METHOD SetUserFrame : BOOL
VAR_INPUT
	Frame	: ST_CartesianPoint;
END_VAR
VAR_OUTPUT
	task	: RoboConnect.I_Task;
END_VAR
VAR 
  commandString : T_Maxstring; 
  
  tableString : STRING := '{,,,,,}';
END_VAR
// TODO better ways of doing this.
tableString := INSERT(tableString, LREAL_TO_STRING(Frame.c),6);
tableString := INSERT(tableString, LREAL_TO_STRING(Frame.b),5);
tableString := INSERT(tableString, LREAL_TO_STRING(Frame.a),4);
tableString := INSERT(tableString, LREAL_TO_STRING(Frame.z),3);
tableString := INSERT(tableString, LREAL_TO_STRING(Frame.y),2);
tableString := INSERT(tableString, LREAL_TO_STRING(Frame.x),1);

IF NOT commandConstructor.setTool(index := 1, table := tableString, commandOutput => commandString) THEN
	SetUserFrame := FALSE;
  LogWarning('Failed to create command SetUserFrame');
	RETURN;
  
END_IF

SetUserFrame := CallRobotApi_NormalPriority(commandString, task => task);
END_METHOD

METHOD PUBLIC ClearQueue
connection.ClearQueue();
END_METHOD

METHOD Connect
VAR_INPUT
  ip : T_IPv4Addr;
  timeout : TIME;
END_VAR
connection.Connect(ip, V3_Ports.DASHBOARD, timeout);
LogDebug('Connect called');
END_METHOD

METHOD Disconnect
connection.Disconnect();
END_METHOD

METHOD FreeAllTasks
connection.FreeAllTasks();
END_METHOD

METHOD SetRobotType : BOOL
VAR_INPUT
	model : E_DobotTypes;
END_VAR
SetRobotType := connection.SetRobotType(model);
END_METHOD

METHOD PRIVATE CallRobotApi : BOOL
VAR_INPUT
  commandString : DOBOT_CMD_STRING;
  priority : E_CommandPriority;
END_VAR
VAR_OUTPUT
	task	: RoboConnect.I_Task;
END_VAR
CallRobotApi := 
  connection.CallRobotApi(
    commandString := commandString, 
    priority := priority, 
    task => task
  );
END_METHOD

METHOD PRIVATE CallRobotApi_NormalPriority : BOOL
VAR_INPUT
  commandString : DOBOT_CMD_STRING;
END_VAR
VAR_OUTPUT
	task	: RoboConnect.I_Task;
END_VAR
CallRobotApi_NormalPriority := 
  CallRobotApi(
    commandString := commandString, 
    priority := E_CommandPriority.NORMAL, 
    task => task
  );
END_METHOD

{attribute 'monitoring' := 'variable'}
PROPERTY Connected : BOOL
GET
Connected := connection.Connected;
END_GET
END_PROPERTY

{attrribute 'monitoring' := 'variable'}
PROPERTY DobotType : E_DobotTypes
GET
DobotType := connection.DobotType;
END_GET
END_PROPERTY

END_FUNCTION_BLOCK

// V3_API/T_V3CommandAndFeedbackBaseClass
FUNCTION_BLOCK INTERNAL T_V3CommandAndFeedbackBaseClass EXTENDS T_NamedBase
VAR
  commandInvoker : T_CommandInvoker;
  commandQueue : T_CommandQueue;
  taskPool : T_CommandTaskPoolV3;
  tempTask : I_CommandTask;
  commandConstructor : T_DobotCommandConstructor; 
  socket : T_ConnectionTCPIP;
  ip : T_IPv4Addr;
  _dobotType : E_DobotTypes;

  state, prevState : (
    NONE,
    INIT,
    
    DISCONNECTED,
    CONNECTING,
    CONNECTED_STATE,
    DISCONNECTING );

END_VAR
VAR CONSTANT

  AXIS_ONE : INT := 1;
  AXIS_TWO : INT := 2;
  AXIS_THREE : INT := 3;
  AXIS_FOUR : INT := 4;
  AXIS_FIVE : INT := 5;
  AXIS_SIX : INT := 6;

  CART_X : INT := 1;
  CART_Y : INT := 2;
  CART_Z : INT := 3;
  CART_Rx : INT := 4;
  CART_Ry : INT := 5;
  CART_Rz : INT := 6;
END_VAR

socket.CyclicLogic();

CASE state OF

  NONE:
    StateChanged();
    state := INIT;

  INIT:
    IF StateChanged() THEN
      commandInvoker.Initialise(commandQueue);
    END_IF;

    IF _dobotType <> E_DobotTypes.NONE THEN
      state := DISCONNECTED;
    END_IF

  DISCONNECTED:
    StateChanged();

  CONNECTING:
    StateChanged();

    IF socket.IsConnected THEN
      state := CONNECTED_STATE;
    END_IF

  CONNECTED_STATE:
    StateChanged();

    commandInvoker.CyclicLogic();

    IF socket.IsErrorConnect THEN
      LogError('Error connecting');
      Disconnect();
    END_IF

  DISCONNECTING:
    StateChanged();

    IF NOT socket.IsConnected THEN
      state := DISCONNECTED;
    END_IF

END_CASE

METHOD PRIVATE StateChanged : BOOL
StateChanged := prevState <> state;
prevState := state;
END_METHOD

{attribute 'monitoring' := 'variable'}
PROPERTY Connected : BOOL
GET
Connected := 
  socket.IsConnected 
  AND state = CONNECTED_STATE;
END_GET
END_PROPERTY

{attrribute 'monitoring' := 'variable'}
PROPERTY INTERNAL DobotType : E_DobotTypes
GET
DobotType := _dobotType;
END_GET
END_PROPERTY

METHOD PUBLIC CallRobotApi : BOOL
VAR_INPUT
  commandString : DOBOT_CMD_STRING;
  priority : E_CommandPriority;
END_VAR
VAR_OUTPUT
	task	: RoboConnect.I_Task;
END_VAR
VAR
  tempTask : I_CommandTask;
END_VAR
IF NOT taskPool.GetTask(result => tempTask) THEN
	LogError('No Spare tasks to use from task pool');
	RETURN;
END_IF

tempTask.Initalise(socket,commandstring);
task := tempTask;
commandQueue.AddWithPriority(task, priority);
END_METHOD

METHOD PUBLIC ClearQueue
commandQueue.Clear();
END_METHOD

METHOD Connect : BOOL
VAR_INPUT
  ip : T_IPv4Addr;
  port : UINT;
  timeout : TIME;
END_VAR
IF Connected THEN
  LogWarning('Cannot Connect() as Connected');
  RETURN;

END_IF

socket.Connect(ip := ip, port := port, timeout := timeout);
state := CONNECTING;
Connect := TRUE;
END_METHOD

METHOD Disconnect
socket.Disconnect();
commandInvoker.Reset();
state := DISCONNECTING;
END_METHOD

METHOD FreeAllTasks
taskPool.FreeAllTasks();
END_METHOD

METHOD PRIVATE Initialise : BOOl
VAR_INPUT
  degreesOfFreedom : USINT;
END_VAR
Initialise := commandInvoker.Initialise(commandQueue);
LogInfo('Initialise called');
END_METHOD

METHOD SetRobotType : BOOL
VAR_INPUT
	model : E_DobotTypes;
END_VAR
IF _dobotType <> E_DobotTypes.NONE THEN
  LogDebug('Cannot SetDegreesOfFreedom as already set ');
  RETURN;
  
END_IF

_dobotType := model;
LogDebug(CONCAT('degrees of freedom set to ', TO_STRING(_dobotType)));

SetRobotType := TRUE;
END_METHOD

END_FUNCTION_BLOCK

// V3_API/T_FeedbackV3
FUNCTION_BLOCK T_FeedbackV3 EXTENDS T_Namedbase
VAR
  socket : T_ConnectionTCPIP;
  _ip : T_MaxString;
  _v3DobotFeedBack : DobotCR3Feedback;

  accumulatorArray : ARRAY[1.. ACCUMULATOR_ARRAY_SIZE] OF BYTE;
  fdBkBuffer : ARRAY[0..DOBOT_FDBK_DATA_SIZE] OF BYTE;
  accumulatorIndex: UDINT := 1;
  task : T_Task;
  isFirst : BOOL := TRUE;
  lastPacketReceivedMs : LINT;
  timeSinceLastPacketMs : LINT;
  _timeoutInMs : LINT;
END_VAR
VAR CONSTANT
  MSG_SIZE_BYTE_ZERO_VALUE : USINT := 160;
  MSG_SIZE_BYTE_ONE_VALUE : USINT := 5;
  ACCUMULATOR_ARRAY_SIZE : UDINT := RoboConnect.RoboConnectParams.receiveBufferSize * 4;
  DOBOT_FDBK_DATA_SIZE : UDINT := 1440;
  
END_VAR

IF F_Gate(isFirst) THEN
  task.SetToThisTask();
END_IF

socket.CyclicLogic();
timeSinceLastPacketMs := task.DistributedClockTimeInMs - lastPacketReceivedMs;

IF connected THEN
  CyclicReadFeedback();

  IF timeSinceLastPacketMs > _timeoutInMs THEN
    LogError('Disconnect, as no feedback received within timeout');
    Disconnect();
  END_IF
  
END_IF

METHOD PRIVATE ClearAccumulator
accumulatorIndex := 1;
MEMSET(ADR(accumulatorArray[1]), 0, SIZEOF(accumulatorArray));
END_METHOD

METHOD Connect 
VAR_INPUT
  ip : T_IPv4Addr;
  timeout : TIME;
END_VAR
socket.Connect(ip, V3_Ports.FEEDBACK, timeout);
LogDebug('Connecting');

_timeoutInMs := TO_LINT(timeout); 

lastPacketReceivedMs := task.DistributedClockTimeInMs;
END_METHOD

METHOD CyclicReadFeedback : BOOL // TRUE - new message
VAR
  rcvArray : RoboConnect.RecvBuffer;
  receiveLength : UDINT;
  i, j, arrIndex, decodeIndex : UDINT;
END_VAR

VAR CONSTANT
  ROBOT_TYPE_BYTE_POSITION : INT := 1031;
  NO_ROBOT_TYPE : BYTE := 0;
END_VAR
IF NOT socket.Receive(data => rcvArray, receiveLength => receiveLength) THEN
  RETURN;
END_IF

IF receiveLength = 0 THEN
  RETURN;
END_IF

IF receiveLength + accumulatorIndex > ACCUMULATOR_ARRAY_SIZE THEN
  // No chance of a packet at this point, 
  ClearAccumulator();
END_IF

MEMCPY(destAddr := ADR(accumulatorArray[accumulatorIndex]), srcAddr := ADR(rcvArray[1]), n := receiveLength);

accumulatorIndex := accumulatorIndex + receiveLength;

IF accumulatorIndex <= DOBOT_FDBK_DATA_SIZE THEN
  RETURN;

END_IF

FOR decodeIndex := 1 TO accumulatorIndex - DOBOT_FDBK_DATA_SIZE DO

  IF accumulatorArray[decodeIndex] = MSG_SIZE_BYTE_ZERO_VALUE AND accumulatorArray[decodeIndex + 1] = MSG_SIZE_BYTE_ONE_VALUE THEN

    CyclicReadFeedback := TRUE;

    // get data chunk we want into our fdBkBuffer (a full packet of Dobot FdBk)
    MEMCPY(
        destAddr := ADR(fdBkBuffer[0]),
        srcAddr := ADR(accumulatorArray[decodeIndex]),
        n := DOBOT_FDBK_DATA_SIZE
      );

    accumulatorIndex := AdvanceAccumulatorArray(IndexToAdvanceFrom := decodeIndex + DOBOT_FDBK_DATA_SIZE);
    EXIT;

  END_IF

END_FOR

IF NOT CyclicReadFeedback THEN
  RETURN;

END_IF

//check if cr robot type is valid 
IF fdBkBuffer[ROBOT_TYPE_BYTE_POSITION] = NO_ROBOT_TYPE THEN
  MEMSET(ADR(fdBkBuffer), 0, SIZEOF(fdBkBuffer));

  RETURN;

END_IF

lastPacketReceivedMs := task.DistributedClockTimeInMs;

DecodeFeedback();
END_METHOD

METHOD Disconnect
socket.Disconnect();
LogInfo('Disconnecting');
END_METHOD

METHOD PRIVATE AdvanceAccumulatorArray : UDINT // returns new accumulator index
VAR_INPUT
  IndexToAdvanceFrom : UDINT; // data at this index will be at the first array positon.
END_VAR
IF NOT ByteArrayAdvanceAndClearRemaining(
    arrayToPass := accumulatorArray,
    positionToAdvanceFrom := IndexToAdvanceFrom
  ) THEN

  LogWarning('AdvanceAccumulatorArray failed, accumulatorIndex unchanged');
  AdvanceAccumulatorArray := accumulatorIndex;
  RETURN;

END_IF

AdvanceAccumulatorArray := accumulatorIndex - (IndexToAdvanceFrom - 1);
END_METHOD

METHOD DecodeFeedback : BOOL
VAR
  i, j, arrIndex : UDINT;
END_VAR
_v3DobotFeedBack.MessageSize.arrBytesIn[0] := fdBkBuffer[0];
_v3DobotFeedBack.MessageSize.arrBytesIn[1] := fdBkBuffer[1];

arrIndex := 8;

FOR i := 0 TO 7 DO
  _v3DobotFeedBack.DigitalInputs[i] := BYTE_TO_BOOL(fdBkBuffer[arrIndex + i]);
END_FOR

arrIndex := 16;

FOR i := 0 TO 7 DO
  _v3DobotFeedBack.DigitalOutputs[i] := BYTE_TO_BOOL(fdBkBuffer[arrIndex + i]);
END_FOR

arrIndex := 24;

FOR i := 0 TO 7 DO
  _v3DobotFeedBack.RobotMode.arrBytesIn[i] := fdBkBuffer[arrIndex + i];
END_FOR

arrIndex := 32;

FOR i := 0 TO 7 DO
  _v3DobotFeedBack.TestValue.arrBytesIn[i] := fdBkBuffer[arrIndex + i];
END_FOR

arrIndex := 64;

FOR i := 0 TO 7 DO
  _v3DobotFeedBack.SpeedScaling.arrBytesIn[i] := fdBkBuffer[arrIndex + i];
END_FOR

arrIndex := 72;

FOR i := 0 TO 7 DO
  _v3DobotFeedBack.LinearMomentumNorm.arrBytesIn[i] := fdBkBuffer[arrIndex + i];
END_FOR

arrIndex := 80;

FOR i := 0 TO 7 DO
  _v3DobotFeedBack.VMain.arrBytesIn[i] := fdBkBuffer[arrIndex + i];
END_FOR

arrIndex := 88;

FOR i := 0 TO 7 DO
  _v3DobotFeedBack.VRobot.arrBytesIn[i] := fdBkBuffer[arrIndex + i];
END_FOR

arrIndex := 96;

FOR i := 0 TO 7 DO
  _v3DobotFeedBack.IRobot.arrBytesIn[i] := fdBkBuffer[arrIndex + i];
END_FOR

arrIndex := 120;

FOR j := 0 TO 2 DO
  FOR i := 0 TO 7 DO
    _v3DobotFeedBack.ToolAcceleroMeter[j].arrBytesIn[i] := fdBkBuffer[arrIndex + i];
  END_FOR

  arrIndex := arrIndex + 8;
END_FOR

arrIndex := 144;

FOR j := 0 TO 2 DO
  FOR i := 0 TO 7 DO
    _v3DobotFeedBack.ElbowPosition[j].arrBytesIn[i] := fdBkBuffer[arrIndex + i];
  END_FOR

  arrIndex := arrIndex + 8;
END_FOR

arrIndex := 168;

FOR j := 0 TO 2 DO
  FOR i := 0 TO 7 DO
    _v3DobotFeedBack.ElbowVelocity[j].arrBytesIn[i] := fdBkBuffer[arrIndex + i];
  END_FOR

  arrIndex := arrIndex + 8;
END_FOR

arrIndex := 192;

FOR j := 0 TO 5 DO
  FOR i := 0 TO 7 DO
    _v3DobotFeedBack.QTarget[j].arrBytesIn[i] := fdBkBuffer[arrIndex + i];
  END_FOR

  arrIndex := arrIndex + 8;
END_FOR

arrIndex := 240;

FOR j := 0 TO 5 DO
  FOR i := 0 TO 7 DO
    _v3DobotFeedBack.QDTarget[j].arrBytesIn[i] := fdBkBuffer[arrIndex + i];
  END_FOR

  arrIndex := arrIndex + 8;
END_FOR

arrIndex := 288;

FOR j := 0 TO 5 DO
  FOR i := 0 TO 7 DO
    _v3DobotFeedBack.QDDTarget[j].arrBytesIn[i] := fdBkBuffer[arrIndex + i];
  END_FOR

  arrIndex := arrIndex + 8;
END_FOR

arrIndex := 336;

FOR j := 0 TO 5 DO
  FOR i := 0 TO 7 DO
    _v3DobotFeedBack.ITarget[j].arrBytesIn[i] := fdBkBuffer[arrIndex + i];
  END_FOR

  arrIndex := arrIndex + 8;
END_FOR

arrIndex := 384;

FOR j := 0 TO 5 DO
  FOR i := 0 TO 7 DO
    _v3DobotFeedBack.MTarget[j].arrBytesIn[i] := fdBkBuffer[arrIndex + i];
  END_FOR

  arrIndex := arrIndex + 8;
END_FOR

arrIndex := 432;

FOR j := 0 TO 5 DO
  FOR i := 0 TO 7 DO
    _v3DobotFeedBack.QActual[j].arrBytesIn[i] := fdBkBuffer[arrIndex + i];
  END_FOR

  arrIndex := arrIndex + 8;
END_FOR

arrIndex := 480;

FOR j := 0 TO 5 DO
  FOR i := 0 TO 7 DO
    _v3DobotFeedBack.QDActual[j].arrBytesIn[i] := fdBkBuffer[arrIndex + i];
  END_FOR

  arrIndex := arrIndex + 8;
END_FOR

arrIndex := 528;

FOR j := 0 TO 5 DO
  FOR i := 0 TO 7 DO
    _v3DobotFeedBack.IActual[j].arrBytesIn[i] := fdBkBuffer[arrIndex + i];
  END_FOR

  arrIndex := arrIndex + 8;
END_FOR

arrIndex := 576;

FOR j := 0 TO 5 DO
  FOR i := 0 TO 7 DO
    _v3DobotFeedBack.ActualTCPForce[j].arrBytesIn[i] := fdBkBuffer[arrIndex + i];
  END_FOR

  arrIndex := arrIndex + 8;
END_FOR

arrIndex := 624;

FOR j := 0 TO 5 DO
  FOR i := 0 TO 7 DO
    _v3DobotFeedBack.ToolVectorActual[j].arrBytesIn[i] := fdBkBuffer[arrIndex + i];
  END_FOR

  arrIndex := arrIndex + 8;
END_FOR

arrIndex := 672;

FOR j := 0 TO 5 DO
  FOR i := 0 TO 7 DO
    _v3DobotFeedBack.TCPSpeedActual[j].arrBytesIn[i] := fdBkBuffer[arrIndex + i];
  END_FOR

  arrIndex := arrIndex + 8;
END_FOR

arrIndex := 720;

FOR j := 0 TO 5 DO
  FOR i := 0 TO 7 DO
    _v3DobotFeedBack.TCPForce[j].arrBytesIn[i] := fdBkBuffer[arrIndex + i];
  END_FOR

  arrIndex := arrIndex + 8;
END_FOR

arrIndex := 768;

FOR j := 0 TO 5 DO
  FOR i := 0 TO 7 DO
    _v3DobotFeedBack.ToolVectorTarget[j].arrBytesIn[i] := fdBkBuffer[arrIndex + i];
  END_FOR

  arrIndex := arrIndex + 8;
END_FOR

arrIndex := 816;

FOR j := 0 TO 5 DO
  FOR i := 0 TO 7 DO
    _v3DobotFeedBack.TCPSpeedTarget[j].arrBytesIn[i] := fdBkBuffer[arrIndex + i];
  END_FOR

  arrIndex := arrIndex + 8;
END_FOR

arrIndex := 864;

FOR j := 0 TO 5 DO
  FOR i := 0 TO 7 DO
    _v3DobotFeedBack.MotorTemperatures[j].arrBytesIn[i] := fdBkBuffer[arrIndex + i];
  END_FOR

  arrIndex := arrIndex + 8;
END_FOR

arrIndex := 912;

FOR j := 0 TO 5 DO
  FOR i := 0 TO 7 DO
    _v3DobotFeedBack.JointModes[j].arrBytesIn[i] := fdBkBuffer[arrIndex + i];
  END_FOR

  arrIndex := arrIndex + 8;
END_FOR

arrIndex := 960;

FOR j := 0 TO 5 DO
  FOR i := 0 TO 7 DO
    _v3DobotFeedBack.VActual[j].arrBytesIn[i] := fdBkBuffer[arrIndex + i];
  END_FOR

  arrIndex := arrIndex + 8;
END_FOR

arrIndex := 1008;

FOR i := 0 TO 3 DO
  _v3DobotFeedBack.HandType[i] := fdBkBuffer[arrIndex + i];
END_FOR

_v3DobotFeedBack.User := fdBkBuffer[1012];
_v3DobotFeedBack.Tool.arrBytesIn[0] := fdBkBuffer[1013];
_v3DobotFeedBack.RunQueuedCmd := BYTE_TO_BOOL(fdBkBuffer[1014]);
_v3DobotFeedBack.PauseCmdFlag := BYTE_TO_BOOL(fdBkBuffer[1015]);
_v3DobotFeedBack.VelocityRatio := BYTE_TO_REAL(fdBkBuffer[1016]);
_v3DobotFeedBack.AccelerationRatio := BYTE_TO_REAL(fdBkBuffer[1017]);
_v3DobotFeedBack.JerkRatio := BYTE_TO_REAL(fdBkBuffer[1018]);
_v3DobotFeedBack.XYZVelocityRatio := BYTE_TO_REAL(fdBkBuffer[1019]);
_v3DobotFeedBack.RVelocityRatio := BYTE_TO_REAL(fdBkBuffer[1020]);
_v3DobotFeedBack.XYZAccelerationRatio := BYTE_TO_REAL(fdBkBuffer[1021]);
_v3DobotFeedBack.RAccelerationRatio := BYTE_TO_REAL(fdBkBuffer[1022]);
_v3DobotFeedBack.XYZJerkRatio := BYTE_TO_REAL(fdBkBuffer[1023]);
_v3DobotFeedBack.RJerkRatio := BYTE_TO_REAL(fdBkBuffer[1024]);
_v3DobotFeedBack.BrakeStatus := BYTE_TO_BOOL(fdBkBuffer[1025]);
_v3DobotFeedBack.EnableStatus := BYTE_TO_BOOL(fdBkBuffer[1026]);
_v3DobotFeedBack.DragStatus := BYTE_TO_BOOL(fdBkBuffer[1027]);
_v3DobotFeedBack.RunningStatus := BYTE_TO_BOOL(fdBkBuffer[1028]);
_v3DobotFeedBack.ErrorStatus := BYTE_TO_BOOL(fdBkBuffer[1029]);
_v3DobotFeedBack.JogStatusCR := BYTE_TO_BOOL(fdBkBuffer[1030]);
_v3DobotFeedBack.CRRobotType := BYTE_TO_INT(fdBkBuffer[1031]);
_v3DobotFeedBack.DragButtonSignal := BYTE_TO_BOOL(fdBkBuffer[1032]);
_v3DobotFeedBack.EnableButtonSignal := BYTE_TO_BOOL(fdBkBuffer[1033]);
_v3DobotFeedBack.RecordButtonSignal := BYTE_TO_BOOL(fdBkBuffer[1034]);
_v3DobotFeedBack.ReappearButtonSignal := BYTE_TO_BOOL(fdBkBuffer[1035]);
_v3DobotFeedBack.JawButtonSignal := BYTE_TO_BOOL(fdBkBuffer[1036]);
_v3DobotFeedBack.SixForceOnline := BYTE_TO_BOOL(fdBkBuffer[1037]);

arrIndex := 1120;

FOR j := 0 TO 5 DO
  FOR i := 0 TO 7 DO
    _v3DobotFeedBack.MActual[j].arrBytesIn[i] := fdBkBuffer[arrIndex + i];
  END_FOR

  arrIndex := arrIndex + 8;
END_FOR

_v3DobotFeedBack.Load[0] := BYTE_TO_REAL(fdBkBuffer[1168]);
_v3DobotFeedBack.Load[1] := BYTE_TO_REAL(fdBkBuffer[1176]);
_v3DobotFeedBack.Load[2] := BYTE_TO_REAL(fdBkBuffer[1184]);
_v3DobotFeedBack.Load[3] := BYTE_TO_REAL(fdBkBuffer[1192]);
_v3DobotFeedBack.Load[4] := BYTE_TO_REAL(fdBkBuffer[1296]);

arrIndex := 1304;

FOR j := 0 TO 5 DO
  FOR i := 0 TO 7 DO
    _v3DobotFeedBack.SixForceValue[j].arrBytesIn[i] := fdBkBuffer[arrIndex + i];
  END_FOR

  arrIndex := arrIndex + 8;
END_FOR

arrIndex := 1352;

FOR j := 0 TO 3 DO
  FOR i := 0 TO 7 DO
    _v3DobotFeedBack.TargetQuaternion[j].arrBytesIn[i] := fdBkBuffer[arrIndex + i];
  END_FOR

  arrIndex := arrIndex + 8;
END_FOR

arrIndex := 1384;

FOR j := 0 TO 3 DO
  FOR i := 0 TO 7 DO
    _v3DobotFeedBack.ActualQuaternion[j].arrBytesIn[i] := fdBkBuffer[arrIndex + i];
  END_FOR

  arrIndex := arrIndex + 8;
END_FOR
END_METHOD

{attribute 'monitoring' := 'variable'}
PROPERTY Connected : BOOL
GET
Connected := socket.IsConnected;
END_GET
END_PROPERTY

{attribute 'monitoring' := 'variable'}
PROPERTY Error : BOOL
GET
Error := socket.IsErrorConnect or socket.IsErrorReceive;
END_GET
END_PROPERTY

{attribute 'monitoring' := 'variable'}
PROPERTY ErrorID : LREAL
GET
ErrorID := socket.ErrID;
END_GET
END_PROPERTY

PROPERTY PUBLIC RobotFdBack : REFERENCE TO DobotCR3Feedback
GET
RobotFdBack REF= _v3DobotFeedBack;
END_GET
SET
END_SET
END_PROPERTY

END_FUNCTION_BLOCK

// V3_API/T_MotionV3
FUNCTION_BLOCK T_MotionV3 EXTENDS T_NamedBase
VAR
  CartesianDynamics : RoboConnect.ST_CartesianPoint;
  connection : T_V3CommandAndFeedbackBaseClass;
  commandConstructor : T_DobotCommandConstructor;
  tempTask : RoboConnect.I_task;
END_VAR
VAR CONSTANT
  AXIS_ONE : INT := 1;
  AXIS_TWO : INT := 2;
  AXIS_THREE : INT := 3;
  AXIS_FOUR : INT := 4;
  AXIS_FIVE : INT := 5;
  AXIS_SIX : INT := 6;

  CART_X : INT := 1;
  CART_Y : INT := 2;
  CART_Z : INT := 3;
  CART_Rx : INT := 4;
  CART_Ry : INT := 5;
  CART_Rz : INT := 6;
END_VAR

connection();

METHOD PUBLIC ClearQueue
connection.ClearQueue();
END_METHOD

METHOD Connect 
VAR_INPUT
  ip : T_IPv4Addr;
  timeout : TIME;
END_VAR
connection.Connect(ip, V3_Ports.MOTION, timeout);
LogDebug('Connect called');
END_METHOD

METHOD Disconnect
connection.Disconnect();
END_METHOD

METHOD FreeAllTasks
connection.FreeAllTasks();
END_METHOD

METHOD JogCartesian : BOOL
VAR_INPUT
	AxisIndex	: INT;
	AxisDirection	: BOOL;
END_VAR
VAR_OUTPUT
	task	: RoboConnect.I_Task;
END_VAR
VAR 
  commandString : T_Maxstring;
  targetJogAxis : ARRAY[0..6] OF STRING := ['','X', 'Y', 'Z', 'Rx', 'Ry', 'Rz'];
END_VAR
IF AxisIndex = CART_X THEN
	IF CartesianDynamics.x = 0 THEN
		JogCartesian := FALSE; 
		RETURN;
	END_IF
ELSIF AxisIndex = CART_Y THEN
	IF CartesianDynamics.y = 0 THEN
		JogCartesian := FALSE; 
		RETURN;
	END_IF
ELSIF AxisIndex = CART_Z THEN
	IF CartesianDynamics.z = 0 THEN
		JogCartesian := FALSE; 
		RETURN;
	END_IF
ELSIF AxisIndex = CART_Rx THEN
	IF CartesianDynamics.a = 0 THEN
		JogCartesian := FALSE; 
		RETURN;
	END_IF
ELSIF AxisIndex = CART_Ry THEN
	IF CartesianDynamics.b = 0 THEN
		JogCartesian := FALSE; 
		RETURN;
	END_IF
ELSIF AxisIndex = CART_Rz THEN
	IF CartesianDynamics.c = 0 THEN
		JogCartesian := FALSE; 
		RETURN;
	END_IF
END_IF


IF NOT commandConstructor.MoveJogCartesian(axisID := targetJogAxis[AxisIndex], axisDirection := AxisDirection, commandOutput => commandString) THEN
	JogCartesian := FALSE;
	RETURN;
END_IF

JogCartesian := CallRobotApi(commandString, E_CommandPriority.NORMAL, task => task);
END_METHOD

METHOD JogJointAxis : BOOL
VAR_INPUT
	AxisIndex	: UDINT;
	AxisDirection	: BOOL;
END_VAR
VAR_OUTPUT
	task	: RoboConnect.I_Task;
END_VAR
VAR 
  commandString : DOBOT_CMD_STRING;
END_VAR
IF NOT commandConstructor.MoveJogJointAxis(axisID := AxisIndex, axisDirection := AxisDirection, commandOutput => commandString) THEN
  JogJointAxis := FALSE;
  LogWarning('Failed to create command JogJointAxis');
	RETURN;
  
END_IF

JogJointAxis := CallRobotApi_NormalPriority(commandString, task => task);
END_METHOD

METHOD MoveAbs : BOOL
VAR_INPUT
	point	: RoboConnect.ST_CartesianPoint;
END_VAR
VAR_OUTPUT
	task	: RoboConnect.I_Task;
END_VAR
VAR 
  commandString : T_Maxstring;
END_VAR
{warning disable C0197}
IF NOT commandConstructor.MovL(
    x := point.x,
    y := point.y,
    z := point.z,
    rX := point.a,
    rY := point.b,
    rZ := point.c,
    commandOutput => commandString
  ) THEN
  MoveAbs := FALSE;
  LogWarning('Failed to create command MoveAbs');
	RETURN;
  
END_IF
{warning restore C0197}

MoveAbs := CallRobotApi_NormalPriority(commandString, task => task);
END_METHOD

METHOD MoveJ : BOOL
VAR_IN_OUT
	joints : ARRAY[*] OF LREAL;
END_VAR
VAR_OUTPUT
	task	: RoboConnect.I_Task;
END_VAR
VAR 
  commandString : T_Maxstring;
  lower, upper, arrSize, i, indexOffset : DINT;
  jointsToSend :  ARRAY[1..6] OF LREAL;
END_VAR
lower :=  LOWER_BOUND(joints, 1);
upper :=  UPPER_BOUND(joints, 1);

arrSize := (upper - lower) + 1;

IF arrSize < 4 OR arrSize > 6 THEN
  LogError(CONCAT('MovJ array size is invalid: ', TO_STRING(arrSize)));
  MoveJ := FALSE;
  RETURN;
  
END_IF

indexOffset := 1 - lower;
FOR i := lower TO upper DO
  jointsToSend[i + indexOffset] := joints[i];
  
END_FOR

{warning disable C0197}
IF NOT commandConstructor.JointMovJ(
  jointsToSend[1],
  jointsToSend[2],
  jointsToSend[3],
  jointsToSend[4],
  jointsToSend[5],
  jointsToSend[6],
  commandOutput => commandString
) THEN
  MoveJ := FALSE;
  LogWarning('Failed to create command MoveJ');
  RETURN;

END_IF

MoveJ := CallRobotApi_NormalPriority(commandString, task => task);
END_METHOD

METHOD SetRobotType : BOOL
VAR_INPUT
	model : E_DobotTypes;
END_VAR
SetRobotType := 
  connection.SetRobotType(model := model);
END_METHOD

METHOD PRIVATE CallRobotApi : BOOL
VAR_INPUT
  commandString : DOBOT_CMD_STRING;
  priority : E_CommandPriority;
END_VAR
VAR_OUTPUT
	task	: RoboConnect.I_Task;
END_VAR
CallRobotApi := 
  connection.CallRobotApi(
    commandString := commandString, 
    priority := priority, 
    task => task
  );
END_METHOD

METHOD PRIVATE CallRobotApi_NormalPriority : BOOL
VAR_INPUT
  commandString : DOBOT_CMD_STRING;
END_VAR
VAR_OUTPUT
	task	: RoboConnect.I_Task;
END_VAR
CallRobotApi_NormalPriority := 
  connection.CallRobotApi(
    commandString := commandString, 
    priority := E_CommandPriority.NORMAL, 
    task => task
  );
END_METHOD

{attribute 'monitoring' := 'variable'}
PROPERTY Connected : BOOL
GET
Connected := connection.Connected;
END_GET
END_PROPERTY

{attrribute 'monitoring' := 'variable'}
PROPERTY DobotType : E_DobotTypes
GET
DobotType := connection.DobotType;
END_GET
END_PROPERTY

END_FUNCTION_BLOCK

// T_DobotV3_Cr_Nova
FUNCTION_BLOCK T_DobotV3_Cr_Nova EXTENDS T_Namedbase IMPLEMENTS I_RoboConnect
VAR
  dashboard : T_DashboardV3;
  feedback : T_FeedbackV3;
  motion : T_MotionV3;

  _ip : T_MaxString;

  state, prevState : (INIT,
    IDLE,
    CONNECTING,
    READY,
    DISCONNECTING,
    ERROR_STATE);

  initInvoker : BOOL;

  numberOfAxes : UDINT := 6;

  cartesianDynamics : RoboConnect.ST_CartesianPoint;
  cartAtPosDeltas : RoboConnect.ST_CartesianPoint := (
    x := 1,
    y := 1.0,
    z := 1.0,
    a := 0.1,
    b := 0.1,
    c := 0.1
  );
  
  jointAtPosDeltas : ARRAY[1..6] OF LREAL := [0.1, 0.1, 0.1, 0.1, 0.1, 0.1];
  realTimeFeedback : DobotCR3Feedback;

END_VAR

METHOD GetAnalogOutput : BOOL
VAR_INPUT
	Index	: UINT;
END_VAR
VAR_OUTPUT
	task	: RoboConnect.I_NumberResultTask;
END_VAR
END_METHOD

METHOD GetAxisCurrents : BOOL
VAR_IN_OUT
  Values : ARRAY[*] OF LREAL;
END_VAR
VAR_OUTPUT
  task : I_Task;
END_VAR
VAR 
	valuesIndexer : INT;
END_VAR
FOR valuesIndexer := 0 TO SIZEOF(values) DO
	Values[valuesIndexer] := realTimeFeedback.IActual[valuesIndexer].realOut;
END_FOR

GetAxisCurrents := TRUE;
END_METHOD

METHOD GetAxisPositions : BOOL
VAR_IN_OUT
  Values : ARRAY[*] OF LREAL;
END_VAR
VAR_OUTPUT
  task : I_Task;
END_VAR
VAR 
	valuesIndexer : INT;
END_VAR
FOR valuesIndexer := 0 TO SIZEOF(Values) DO 
	values[valuesIndexer] := realTimeFeedback.QActual[valuesIndexer].realOut;
END_FOR
GetAxisPositions := true;
END_METHOD

METHOD GetAxisTemperatures : BOOL
VAR_IN_OUT
  Values : ARRAY[*] OF LREAL;
END_VAR
VAR_OUTPUT
  task : I_Task;
END_VAR
VAR 
	valuesIndexer : INT;
END_VAR
FOR valuesIndexer := 0 TO SIZEOF(Values) DO
	Values[valuesIndexer] := realTimeFeedback.MotorTemperatures[valuesIndexer].realOut;
END_FOR

GetAxisTemperatures := TRUE;
END_METHOD

METHOD GetDigitalOutput : BOOL
VAR_INPUT
	Index	: UINT;
END_VAR
VAR_OUTPUT
	task	: RoboConnect.I_BoolResultTask;
	value 	: BOOL;
END_VAR
value := realTimeFeedback.DigitalOutputs[Index];
GetDigitalOutput := TRUE;
END_METHOD

METHOD GetToolAnalogOutput : BOOL
VAR_INPUT
	Index	: UINT;
END_VAR
VAR_OUTPUT
	task	: RoboConnect.I_NumberResultTask;
END_VAR
END_METHOD

METHOD GetToolDigitalOutput : BOOL
VAR_INPUT
	Index	: UINT;
END_VAR
VAR_OUTPUT
	task	: RoboConnect.I_BoolResultTask;
END_VAR
END_METHOD

METHOD ClearError : BOOL
VAR_OUTPUT
	task	: RoboConnect.I_Task;
END_VAR
ClearError := dashboard.ClearError(task => task);
END_METHOD

METHOD Connect : BOOL
state := CONNECTING;
END_METHOD

METHOD CyclicLogic
motion();
dashboard();
feedback();

CASE state OF
  INIT:

    IF StateChanged() THEN
      state := IDLE;

    END_IF

  IDLE:
  // WAIT

  CONNECTING:
    IF StateChanged() THEN
      feedback.Connect(_ip, timeout := RoboConnect.RoboConnectParams.TimeOut);
      dashboard.Connect(_ip, timeout := RoboConnect.RoboConnectParams.TimeOut);
      motion.Connect(_ip, timeout := RoboConnect.RoboConnectParams.TimeOut);

    END_IF

    // if timer elapses go to error state and log and set ID to failed to connect

    IF feedback.Connected AND dashboard.Connected AND motion.Connected THEN
      state := Ready;
    END_IF

  READY:

    realTimeFeedback := feedback.RobotFdBack;
    
    IF NOT (feedback.Connected AND dashboard.Connected AND motion.Connected) THEN
      LogWarning('Disconnecting as NOT(feedback.Connected AND dashboard.Connected AND motion.Connected)');
      state := DISCONNECTING;
    END_IF

  DISCONNECTING:
    IF StateChanged() THEN
      feedback.Disconnect();
      dashboard.Disconnect();
      motion.Disconnect();
    END_IF

    IF NOT feedback.Connected AND NOT dashboard.Connected AND NOT motion.Connected THEN
      state := IDLE;
    END_IF

  ERROR_STATE:

END_CASE
END_METHOD

METHOD Disable : BOOL
VAR_OUTPUT
	task	: RoboConnect.I_Task;
END_VAR
Disable := dashboard.Disable(task => task);
END_METHOD

METHOD Disconnect : BOOL
VAR_OUTPUT
	task	: RoboConnect.I_Task;
END_VAR
state := DISCONNECTING;
END_METHOD

METHOD Enable : BOOL
VAR_OUTPUT
	task	: RoboConnect.I_Task;
END_VAR
Enable := dashboard.Enable(task => task);
END_METHOD

METHOD FreeAllTasks
dashboard.FreeAllTasks();
dashboard.ClearQueue();

motion.FreeAllTasks();
motion.ClearQueue();
END_METHOD

METHOD GetJointPositions : BOOL (* false if incompatible array length*)
VAR_IN_OUT
  (* values overwritten with joint positions.*)
  joints : ARRAY[*] OF LREAL; // positions 1..NumberOfAxes will be used. passed array should be dimensioned accordingly
END_VAR
VAR
  lower, upper, ind : DINT;
END_VAR
lower :=  LOWER_BOUND(joints, 1);
upper :=  UPPER_BOUND(joints, 1);
  
IF numberOfAxes = 0 THEN
  LogError('GetJointPositions() : numberOfAxes = 0');
  RETURN;
  
END_IF

GetJointPositions := 
  (lower <= 1)
  AND (upper >= TO_DINT(numberOfAxes));
  
IF NOT GetJointPositions THEN
  RETURN;
  
END_IF

FOR ind := 0 TO TO_DINT(numberOfAxes) -1 DO
  joints[ind + 1] := feedback.RobotFdBack.QActual[ind].realOut;
END_FOR
END_METHOD

METHOD Halt : BOOL
VAR_OUTPUT
	task	: RoboConnect.I_Task;
END_VAR
Halt := dashboard.Halt(task => task);

//IF NOT commandConstructor.pause(commandOutput => commandString) THEN
//	Halt := FALSE;
//	RETURN;
//END_IF

//IF NOT taskList.GetTask(result => tempTask) THEN
//	LogError('No Spare tasks to use from task pool');
//	RETURN;	
//END_IF

//tempTask.Initalise(dashboard, commandstring);
//_commandQueue.AddNormalPriority(temptask);
//Halt := TRUE;
END_METHOD

METHOD IsAtCartesianPosition : BOOL
VAR_INPUT
	point	: RoboConnect.ST_CartesianPoint;
END_VAR
IsAtCartesianPosition :=
 F_IsAtPositionCartesian(
  actual := CartesianPosition,
  target := point,
  delta := cartAtPosDeltas, 
 );
END_METHOD

METHOD IsAtJointPosition : BOOL
VAR_IN_OUT
  joints : ARRAY[*] OF LREAL; // positions 1..NumberOfAxes will be used. passed array should be dimensioned accordingly
END_VAR
VAR
  actJointsPos : ARRAY[1..6] OF LREAL;
  lower, upper, ind : DINT;
END_VAR
GetJointPositions(joints := actJointsPos);

IsAtJointPosition :=
  F_IsAtPositionJoint(
  actual := actJointsPos,
  target := joints,
  delta := jointAtPosDeltas
);
END_METHOD

{warning 'add method implementation '}
METHOD JogAxis : BOOL (* default tool and user frame*)
VAR_INPUT
	(* joint or enumerated cartesian direction/vector. See concrete type docs for enumeration of cartesian coords.*)
	axisIndex	: UDINT;
	(* TRUE = positive, FALSE = negative*)
	axisDirection	: BOOL;
	(* Cartesian or Joint space*)
	jogType	: RoboConnect.E_JogType;
END_VAR
VAR_OUTPUT
	task	: RoboConnect.I_Task;
END_VAR
END_METHOD

{warning 'add method implementation '}
METHOD JogAxisAdvanced : BOOL
VAR_INPUT
	(* joint or enumerated cartesian direction/vector. See concrete type docs for enumeration of cartesian coords.*)
	axisIndex	: UDINT;
	(* TRUE = positive, FALSE = negative*)
	axisDirection	: BOOL;
	(* Cartesian or Joint space*)
	jogType	: RoboConnect.E_JogType;
	(* set to 0 to leave default*)
	coordType	: INT;
	(* set to 0 to leave default*)
	user	: INT;
	(* set to 0 to leave default*)
	tool	: INT;
END_VAR
VAR_OUTPUT
	task	: RoboConnect.I_Task;
END_VAR
END_METHOD

METHOD JogCartesian : BOOL
VAR_INPUT
	AxisIndex	: INT;
	AxisDirection	: BOOL;
END_VAR
VAR_OUTPUT
	task	: RoboConnect.I_Task;
END_VAR
VAR 
  commandString : T_Maxstring;
  targetJogAxis : ARRAY[0..6] OF STRING := ['','X', 'Y', 'Z', 'Rx', 'Ry', 'Rz'];
END_VAR
motion.JogCartesian(AxisIndex, AxisDirection, task => task);

//IF AxisIndex = CART_X THEN
//	IF CartesianDynamics.x = 0 THEN
//		JogCartesian := FALSE; 
//		RETURN;
//	END_IF
//ELSIF AxisIndex = CART_Y THEN
//	IF CartesianDynamics.y = 0 THEN
//		JogCartesian := FALSE; 
//		RETURN;
//	END_IF
//ELSIF AxisIndex = CART_Z THEN
//	IF CartesianDynamics.z = 0 THEN
//		JogCartesian := FALSE; 
//		RETURN;
//	END_IF
//ELSIF AxisIndex = CART_Rx THEN
//	IF CartesianDynamics.a = 0 THEN
//		JogCartesian := FALSE; 
//		RETURN;
//	END_IF
//ELSIF AxisIndex = CART_Ry THEN
//	IF CartesianDynamics.b = 0 THEN
//		JogCartesian := FALSE; 
//		RETURN;
//	END_IF
//ELSIF AxisIndex = CART_Rz THEN
//	IF CartesianDynamics.c = 0 THEN
//		JogCartesian := FALSE; 
//		RETURN;
//	END_IF
//END_IF


//IF NOT commandConstructor.MoveJogCartesian(axisID := targetJogAxis[AxisIndex], axisDirection := AxisDirection, commandOutput => commandString) THEN
//	JogCartesian := FALSE;
//	RETURN;
//END_IF

//IF NOT taskList.GetTask(result => tempTask) THEN
//	LogError('No Spare tasks to use from task pool');
//	JogCartesian := FALSE;
//	RETURN;
//END_IF

//tempTask.Initalise(motion, commandString);
//task := tempTask;
//_commandQueue.AddNormalPriority(temptask);
//JogCartesian := TRUE;
END_METHOD

METHOD JogJointAxis : BOOL
VAR_INPUT
	AxisIndex	: UDINT;
	AxisDirection	: BOOL;
END_VAR
VAR_OUTPUT
	task	: RoboConnect.I_Task;
END_VAR
VAR 
  commandString : DOBOT_CMD_STRING;
END_VAR
JogJointAxis := motion.JogJointAxis(AxisIndex, AxisDirection, task => task);

//IF NOT (NumberOfAxis = 0 OR AxisIndex > NumberOfAxis) THEN
//	IF NOT commandConstructor.MoveJogJointAxis(axisID := AxisIndex, axisDirection := AxisDirection, commandOutput => commandString) THEN
//		JogJointAxis := FALSE;
//		RETURN;
//	END_IF

//	IF NOT taskList.GetTask(result => tempTask) THEN
//  		RETURN;
//	END_IF

//	tempTask.Initalise(motion, commandString);
//	task := tempTask;
//	_commandQueue.AddNormalPriority(temptask);
//	JogJointAxis := TRUE;
//	RETURN;
//ELSE
//  JogJointAxis := FALSE;
//	RETURN;	
//END_IF
END_METHOD

METHOD MoveAbs : BOOL
VAR_INPUT
	point	: RoboConnect.ST_CartesianPoint;
END_VAR
VAR_OUTPUT
	task	: RoboConnect.I_Task;
END_VAR
VAR 
  commandString : T_Maxstring;
END_VAR
MoveAbs := motion.MoveAbs(point, task => task);

//IF NOT commandConstructor.MovJ(
//	x := point.x,
//	y := point.y,
//	z := point.z,
//	rX := point.a,
//	rY := point.b,
//	rZ := point.z,
//	commandOutput => commandString)THEN
//		MoveAbs := FALSE;
//		RETURN;
//END_IF

//IF NOT taskList.GetTask(result => temptask) THEN
//	LogError('No Spare tasks to use from task pool');
//	RETURN;
//END_IF

//tempTask.Initalise(motion,commandString);
//task := tempTask;
//_commandQueue.AddNormalPriority(temptask);
//MoveABS := TRUE;
END_METHOD

METHOD MoveJ : BOOL
VAR_IN_OUT
	joints : ARRAY[*] OF LREAL;
END_VAR
VAR_OUTPUT
	task	: RoboConnect.I_Task;
END_VAR
VAR 
  commandString : T_Maxstring;
END_VAR
MoveJ := motion.MoveJ(joints, task => task);

//IF NOT commandConstructor.JointMovJ(
//	Joints[0],
//	Joints[1],
//	Joints[2],
//	Joints[3],
//	Joints[4],
//	Joints[5],
//	commandOutput => commandString) THEN
//		MoveJ := FALSE;
//		RETURN;
//END_IF

//IF NOT taskList.GetTask(result => temptask) THEN
//	LogError('No Spare tasks to use from task pool');
//	RETURN;
//END_IF

//temptask.Initalise(motion,commandString);
//task := tempTask;
//_commandQueue.AddNormalPriority(temptask);
//MoveJ := TRUE;
END_METHOD

METHOD Reset : BOOL
VAR_OUTPUT
	task	: RoboConnect.I_Task;
END_VAR
VAR
	commandString : T_Maxstring;
END_VAR
Reset := dashboard.Reset(task => task);

//IF NOT commandConstructor.resetRobot(commandOutput => commandString) THEN
//	Reset := FALSE;
//	RETURN;
//END_IF

//IF NOT taskList.GetTask(result => tempTask) THEN
//	LogError('No Spare tasks to use from task pool');
//	RETURN;
//END_IF

//temptask.Initalise(dashboard,commandstring);
//task := tempTask;
//_commandQueue.AddNormalPriority(task);
//Reset := TRUE;
END_METHOD

METHOD SetAtPosDeltas : BOOL
VAR_INPUT
  atPosCartesianDeltas : ST_CartesianPoint;
END_VAR
VAR_IN_OUT
  atPosJointDeltas : ARRAY[*] OF LREAL; // positions 1..NumberOfAxes will be used. passed array should be dimensioned accordingly
END_VAR
VAR
  lower, upper, ind : DINT;
END_VAR
lower :=  LOWER_BOUND (atPosJointDeltas, 1); 
upper :=  UPPER_BOUND (atPosJointDeltas, 1); 

IF lower > 1 OR upper < TO_DINT(numberOfAxes) THEN
  LogError('SetAtPosDeltas() : lower > 1 OR upper < numberOfAxes');
  RETURN;
  
END_IF

cartAtPosDeltas := atPosCartesianDeltas;

FOR ind := 1 TO TO_DINT(numberOfAxes) DO
  jointAtPosDeltas[ind] :=  atPosJointDeltas[ind];
  
END_FOR
END_METHOD

METHOD PRIVATE StateChanged : BOOL
IF state = prevState THEN
	RETURN;
END_IF

StateChanged := TRUE;
prevState := state;
RETURN;
END_METHOD

METHOD Stop : BOOL
VAR_OUTPUT
	task	: RoboConnect.I_Task;
END_VAR
VAR
	commandString : T_Maxstring;
END_VAR
Stop := dashboard.Stop(task => task);

//IF NOT commandConstructor.emergencyStop(commandOutput => commandString) THEN
//	Stop := FALSE;
//	RETURN;
//END_IF

//IF NOT taskList.GetTask(result => temptask) THEN
//	LogError('No Spare tasks to use from task pool');
//	RETURN;
//END_IF

//temptask.Initalise(dashboard,commandstring);
//task := tempTask;
//_commandQueue.AddHighPriority(temptask);
//stop := TRUE;
END_METHOD

{attribute 'monitoring' := 'variable'}
PROPERTY CartesianPosition : RoboConnect.ST_CartesianPoint
GET
CartesianPosition.x := realTimeFeedback.ToolVectorActual[0].realOut;
CartesianPosition.y := realTimeFeedback.ToolVectorActual[1].realOut;
CartesianPosition.z := realTimeFeedback.ToolVectorActual[2].realOut;
CartesianPosition.a := realTimeFeedback.ToolVectorActual[3].realOut;
CartesianPosition.b := realTimeFeedback.ToolVectorActual[4].realOut;
CartesianPosition.c := realTimeFeedback.ToolVectorActual[5].realOut;
END_GET
END_PROPERTY

{attribute 'monitoring' := 'variable'}
PROPERTY Connected : BOOL
GET
Connected := feedback.Connected AND dashboard.Connected AND motion.Connected;
END_GET
END_PROPERTY

{attribute 'monitoring' := 'variable'}
PROPERTY Enabled : BOOL
GET
Enabled := Connected AND realTimeFeedback.EnableStatus;
END_GET
END_PROPERTY

{attribute 'monitoring' := 'variable'}
PROPERTY Error : BOOL
GET
Error := Connected AND realTimeFeedback.ErrorStatus;
END_GET
END_PROPERTY

{attribute 'monitoring' := 'variable'}
PROPERTY ErrorID : LREAL
GET
ErrorId := feedback.ErrorID;
END_GET
END_PROPERTY

{warning 'add property implementation'}
PROPERTY Manufacturer : STRING
GET
PUBLIC
Manufacturer := 'Dobot';
END_GET
END_PROPERTY

{warning 'add property implementation'}
PROPERTY Model : STRING
GET
PUBLIC
Model := TO_STRING(dashboard.DobotType);
END_GET
END_PROPERTY

{attribute 'monitoring' := 'variable'}
PROPERTY Running : BOOL
GET
Running := 
  Connected 
  AND 
    (realTimeFeedback.RunningStatus
      OR realTimeFeedback.JogStatusCR
      OR realTimeFeedback.RobotMode.robotMode = RobotModes.Jogging_State);
END_GET
END_PROPERTY

{attribute 'monitoring' := 'variable'}
PROPERTY ToolPosition : RoboConnect.ST_CartesianPoint
GET
ToolPosition.x := realTimeFeedback.ToolvectorActual[0].realOut;
ToolPosition.y := realTimeFeedback.ToolvectorActual[1].realOut;
ToolPosition.z := realTimeFeedback.ToolvectorActual[2].realOut;
ToolPosition.a := realTimeFeedback.ToolvectorActual[3].realOut;
ToolPosition.b := realTimeFeedback.ToolvectorActual[4].realOut;
ToolPosition.c := realTimeFeedback.ToolvectorActual[5].realOut;
END_GET
END_PROPERTY

METHOD SetAnalogOutput : BOOL
VAR_INPUT
	Index	: UINT;
	Value	: LREAL;
END_VAR
VAR_OUTPUT
	task	: RoboConnect.I_Task;
END_VAR
VAR 
  commandString : T_Maxstring;
END_VAR
SetAnalogOutput := dashboard.SetAnalogOutput(Index, Value, task => task);
END_METHOD

METHOD SetBufferMode : BOOL
VAR_INPUT
	BufferMode	: RoboConnect.E_BufferMode;
END_VAR
SetBufferMode := dashboard.SetBufferMode(BufferMode);
END_METHOD

METHOD SetCarteasianAcceleration : BOOL
VAR_INPUT
	Acceleration	: LREAL;
END_VAR
VAR_OUTPUT
	task	: RoboConnect.I_Task;
END_VAR
SetCarteasianAcceleration := dashboard.SetCarteasianAcceleration(Acceleration, task => task);
END_METHOD

METHOD SetCartesianDynamics : BOOL
VAR_INPUT
	XDynamics : BOOL;
	YDynamics : BOOL;
	ZDynamics : BOOL;
	 
	ADynamics : BOOL;
	BDynamics : BOOL;
	CDynamics : BOOL;
END_VAR
VAR_OUTPUT
  task : I_Task;
END_VAR
SetCartesianDynamics := dashboard.SetCartesianDynamics(
  XDynamics,
	YDynamics, 
	ZDynamics,
	ADynamics, 
	BDynamics, 
	CDynamics, 
  task => task
);
END_METHOD

METHOD SetCartesianSpeed : BOOL
VAR_INPUT
	Speed	: LREAL;
END_VAR
VAR_OUTPUT
	task	: RoboConnect.I_Task;
END_VAR
SetCartesianSpeed := dashboard.SetCartesianSpeed(speed, task => task);
END_METHOD

METHOD SetDigitalOutput : BOOL
VAR_INPUT
	Index	: UINT;
	Value	: BOOL;
END_VAR
VAR_OUTPUT
	task	: RoboConnect.I_Task;
END_VAR
SetDigitalOutput := dashboard.SetDigitalOutput(Index, Value, task => task);
END_METHOD

METHOD SetJointAcceleration : BOOL
VAR_INPUT
	Acceleration	: LREAL;
END_VAR
VAR_OUTPUT
	task	: RoboConnect.I_Task;
END_VAR
SetJointAcceleration := dashboard.SetJointAcceleration(Acceleration, task => task);
END_METHOD

METHOD SetJointSpeed : BOOL
VAR_INPUT
	Speed	: LREAL;
END_VAR
VAR_OUTPUT
	task	: RoboConnect.I_Task;
END_VAR
SetJointSpeed := dashboard.SetJointSpeed(Speed, task => task);
END_METHOD

METHOD SetToolAnalogOutput : BOOL
VAR_INPUT
	Index	: UINT;
	Value	: LREAL;
END_VAR
VAR_OUTPUT
	task	: RoboConnect.I_Task;
END_VAR
SetToolAnalogOutput := dashboard.SetToolAnalogOutput(Index, Value, task => task);
END_METHOD

METHOD SetToolDigitalOutput : BOOL
VAR_INPUT
	Index	: UINT;
	Value	: BOOL;
END_VAR
VAR_OUTPUT
	task	: RoboConnect.I_Task;
END_VAR
VAR 
  commandString : T_Maxstring;
END_VAR
SetToolDigitalOutput := dashboard.SetToolDigitalOutput(Index,Value, task => task);

//IF NOT commandConstructor.tooldo(index := index, STatus := BOOL_TO_INT(Value), commandOutput => commandString) THEN
//	SetToolDigitalOutput := FALSE;
//	RETURN;
//END_IF

//IF NOT taskList.GetTask(result => temptask) THEN
//	LogError('No Spare tasks to use from task pool');
//	RETURN;
//END_IF

//temptask.Initalise(Dashboard,commandString);
//task := tempTask;
//_commandQueue.AddNormalPriority(temptask);
//SetToolDigitalOutput := TRUE;
END_METHOD

METHOD SetToolFrame : BOOL
VAR_INPUT
	Frame	: RoboConnect.ST_CartesianPoint;
END_VAR
VAR_OUTPUT
	task	: RoboConnect.I_Task;
END_VAR
SetToolFrame := dashboard.SetToolFrame(Frame, task => task);

//tableString := INSERT(tableString, LREAL_TO_STRING(Frame.c),6);
//tableString := INSERT(tableString, LREAL_TO_STRING(Frame.b),5);
//tableString := INSERT(tableString, LREAL_TO_STRING(Frame.a),4);
//tableString := INSERT(tableString, LREAL_TO_STRING(Frame.z),3);
//tableString := INSERT(tableString, LREAL_TO_STRING(Frame.y),2);
//tableString := INSERT(tableString, LREAL_TO_STRING(Frame.x),1);
//IF NOT commandConstructor.setTool(index := 1, table := tableString, commandOutput => commandString) THEN
//	setToolFrame := FALSE;
//	RETURN;
//END_IF

//IF NOT taskList.GetTask(result => temptask) THEN
//	LogError('No Spare tasks to use from task pool');
//	RETURN;
//END_IF

//temptask.Initalise(Dashboard,commandString);
//task := tempTask;
//_commandQueue.AddNormalPriority(temptask);
//setToolFrame := TRUE;
END_METHOD

METHOD SetTransitionMode : BOOL
SetTransitionMode := dashboard.SetTransitionMode();
END_METHOD

METHOD SetTransitionParameter : BOOL
VAR_INPUT
	CPratio : LREAL;
END_VAR
VAR_OUTPUT
	task	: RoboConnect.I_Task;
END_VAR
SetTransitionParameter := dashboard.SetTransitionParameter(cPratio, task => task);

//IF  CPratio <100 AND CPratio > 0 THEN
//	IF NOT commandConstructor.cp(ratio := CPratio, commandOutput => commandString) THEN
//		SetTransitionParameter := FALSE;
//		RETURN;
//	END_IF

//	IF NOT taskList.GetTask(result => temptask) THEN
//	LogError('No Spare tasks to use from task pool');
//		RETURN;
//	END_IF

//	temptask.Initalise(Dashboard,commandString);
//	task := tempTask;
//	_commandQueue.AddNormalPriority(temptask);
//	SetTransitionParameter := TRUE;
//ELSE
//	SetTransitionParameter := FALSE;
//END_IF
END_METHOD

METHOD SetUserFrame : BOOL
VAR_INPUT
	Frame	: ST_CartesianPoint;
END_VAR
VAR_OUTPUT
	task	: RoboConnect.I_Task;
END_VAR
VAR 
  commandString : T_Maxstring; 
  
  tableString : STRING := '{,,,,,}';
END_VAR
SetUserFrame := dashboard.SetUserFrame(Frame, task => task);

//tableString := INSERT(tableString, LREAL_TO_STRING(Frame.c),6);
//tableString := INSERT(tableString, LREAL_TO_STRING(Frame.b),5);
//tableString := INSERT(tableString, LREAL_TO_STRING(Frame.a),4);
//tableString := INSERT(tableString, LREAL_TO_STRING(Frame.z),3);
//tableString := INSERT(tableString, LREAL_TO_STRING(Frame.y),2);
//tableString := INSERT(tableString, LREAL_TO_STRING(Frame.x),1);
//IF NOT commandConstructor.setTool(index := 1, table := tableString, commandOutput => commandString) THEN
//	SetUserFrame := FALSE;
//	RETURN;
//END_IF

//IF NOT taskList.GetTask(result => temptask) THEN
//	LogError('No Spare tasks to use from task pool');
//	RETURN;
//END_IF

//temptask.Initalise(Dashboard,commandString);
//task := tempTask;
//_commandQueue.AddNormalPriority(temptask);
//SetUserFrame := TRUE;
END_METHOD

METHOD FB_init : BOOL
VAR_INPUT
	bInitRetains : BOOL; // if TRUE, the retain variables are initialized (warm start / cold start)
	bInCopyCode : BOOL;  // if TRUE, the instance afterwards gets moved into the copy code (online change)
  DobotModel : E_DobotTypes;
END_VAR
dashboard.SetRobotType(DobotModel);
motion.SetRobotType(DobotModel);
END_METHOD

METHOD SetConnectionProperties : BOOL
VAR_INPUT
	Ip : T_MaxString;
END_VAR
_ip := Ip;
SetConnectionProperties := TRUE;
END_METHOD

END_FUNCTION_BLOCK
